PROGRAM MAIN
VAR
	b_YelloPushed : BOOL;
	b_BluePushed : BOOL;
	byte_decider : BYTE;
	i_EdgdetectorYellow : EdgeDetector_1;
	i_EdgdetectorBlue : EdgeDetector_1;
	b_risingEdge : BOOL;
	state : SafeState;
END_VAR

i_EdgdetectorYellow();
i_EdgdetectorYellow.inputValue := GVL.b_buttonYellow;
b_YelloPushed := i_EdgdetectorYellow.riesingEdge;
i_EdgdetectorBlue();
i_EdgdetectorBlue.inputValue := GVL.b_buttonBlue;
b_BluePushed := i_EdgdetectorBlue.riesingEdge;
IF b_YelloPushed OR b_BluePushed THEN
	b_risingEdge := TRUE;
	ELSE
	b_risingEdge := FALSE;
END_IF
CASE state OF
	0 : GVL.bA_CodePins[1] := TRUE;		// State = Init
		GVL.bA_CodePins[2] := FALSE;
		GVL.bA_CodePins[3] := FALSE;
		GVL.bA_CodePins[4] := TRUE;
		state :=1 ;		
	1 : GVL.b_LampeCorrect := FALSE;	// State = Close
		GVL.b_LampeWrong := FALSE;
		GVL.i_correctCounter := 0;
		GVL.i_currentIndex := 1;
		GVL.i_lightDuration := 5000;
		state :=3;		
	2 : IF GVL.i_lightDuration >0 THEN						// State = CorrectCode
		GVL.b_LampeCorrect := TRUE;							// Turn the Green 	
		GVL.i_lightDuration := GVL.i_lightDuration -10;
		ELSE
		GVL.b_LampeCorrect := FALSE;
		state :=1;				// Time is Over > Next state > Close		
		END_IF
	3 : IF b_risingEdge THEN	// State = CheCkDigit
		CASE GVL.i_currentIndex OF
			1 : IF GVL.bA_CodePins[GVL.i_currentIndex] = b_YelloPushed THEN
				GVL.i_currentIndex := GVL.i_currentIndex +1;
				ELSE
					state := 4;	
				END_IF
			2 : IF GVL.bA_CodePins[GVL.i_currentIndex] = NOT b_BluePushed THEN
				GVL.i_currentIndex := GVL.i_currentIndex +1;
				ELSE
					state := 4;	
				END_IF
			3 : IF GVL.bA_CodePins[GVL.i_currentIndex] = NOT b_BluePushed THEN
				GVL.i_currentIndex := GVL.i_currentIndex +1;
				ELSE
					state := 4;	
				END_IF
			4 : IF GVL.bA_CodePins[GVL.i_currentIndex] = b_YelloPushed THEN
					state := 2;	
				ELSE
					state := 4;	
				END_IF		
		END_CASE
		ELSE
		state := 3;		// no button detected > dont change State.
		END_IF
	4 : IF GVL.i_lightDuration >0 THEN						// State = WrongCode
		GVL.b_LampeWrong := TRUE;							// Turn the Red 	
		GVL.i_lightDuration := GVL.i_lightDuration -10;
		ELSE
		GVL.b_LampeWrong := FALSE;
		state :=1;				// Time is Over > Next state > Close		
		END_IF
END_CASE

END_PROGRAM

(* stored: Version 1.1.0.1, ProductVersion 3.1.4022.12
   POU MAIN: Id {575199f3-3758-40d7-b7a6-a55d5906ab45}, SpecialFunc None *)
